INTERFACE ITF_EquipmentBase EXTENDS ITF_Base

PROPERTY AlarmListDetails : Reference to ST_EquipmentAlarmListDetails
GET
END_GET
END_PROPERTY

PROPERTY MainAlarm : Reference to ST_EquipmentAlarm
GET
END_GET
END_PROPERTY

METHOD Reset
END_METHOD

END_INTERFACE

(* stored: Version 1.1.0.1
   Itf ITF_EquipmentBase: Id {4cc029b0-1afe-4c84-800d-5d2f83376e25}
   Property AlarmListDetails: Id {903a1200-548f-46b3-8aa2-58d8db6ebb7c}
   Get Get: Id {79ba21a9-e9f8-4a9e-a4c8-f59b1d2f7c28}
   Property MainAlarm: Id {314f3074-d37f-425f-9578-1f95c292c8db}
   Get Get: Id {0008029c-2913-4a3e-984e-4e30149dd0f3}
   Method Reset: Id {dcbf8e5f-029c-477e-a94f-255c5f675baf} *)
